// Compares value A to generic value B of any type and returns the evaluation.
FUNCTION F_Compare_Any : T_Comparison
VAR_INPUT
	A : ANY;
	B : ANY;
END_VAR

F_Compare_Any := F_Compare_Generics(A, B);

END_FUNCTION

(* stored: Version 1.1.0.1
   POU F_Compare_Any: Id {4016674c-f8d8-0eff-037e-3198817fead0}, SpecialFunc None *)
